// TIA Portal V16 export
// export: Created 2021-07-12T14:47:18.7545958Z, ExportSetting WithDefaults, DisplayName Totally Integrated Automation Portal, DisplayVersion V16, DisplayName TIA Portal Version Control Interface, DisplayVersion V16, DisplayName TIA Portal Openness, DisplayVersion V16, DisplayName STEP 7 Professional, DisplayVersion V16, DisplayName STEP 7 Safety, DisplayVersion V16, DisplayName WinCC Professional, DisplayVersion V16
TYPE "LSimaHydTO_typeSmoothingFilter"
TITLE = LSimaHydTO_typeSmoothingFilter
// Settings of the smoothing filter
// stored: IsFailsafeCompliant false
   STRUCT
      VelocityFilter { S7_SetPoint := 'True'} : LReal := 0.0;   // Time constant for actual velocity smoothing filter [s]
      AccelerationFilter { S7_SetPoint := 'True'} : LReal := 0.0;   // Time constant for actual acceleration smoothing filter [s]
   END_STRUCT;
END_TYPE
